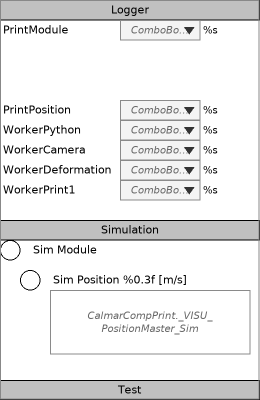
VISUALIZATION _VISU_Pm_Maxliner_Debug  // 260x400
VAR_IN_OUT
	mInst : FB_PrintModule_Maxliner;
END_VAR
    Rectangle (0,220 260x20), "Simulation"
    Ellipse (20,270 20x20), tooltip "Sim position"
        toggle mInst.fbPrintPosition._bSim
    Rectangle (50,270 200x20), "Sim Position %0.3f [m/s]", text variable: mInst.fbPrintPosition.fbPositionMaster._fSimSpeed
        OnMouseClick: write the text variable via Default
    Rectangle (0,0 260x20), "Logger"
    Rectangle (0,100 120x20), "PrintPosition"
    Rectangle (200,100 60x20), "%s", tooltip "LogLevel", text variable: mInst.fbPrintPosition._loglevel
        OnMouseClick: write the text variable via Default
    Rectangle (0,140 120x20), "WorkerCamera"
    Rectangle (200,140 60x20), "%s", tooltip "LogLevel", text variable: mInst.fbWorkerCamera._loglevel
        OnMouseClick: write the text variable via Default
    Rectangle (0,180 120x20), "WorkerPrint1"
    Rectangle (200,180 60x20), "%s", tooltip "LogLevel", text variable: mInst.fbWorkerPrint[1]._loglevel
        OnMouseClick: write the text variable via Default
    Rectangle (0,160 120x20), "WorkerDeformation"
    Rectangle (200,160 60x20), "%s", tooltip "LogLevel", text variable: mInst.fbWorkerDeformation._loglevel
        OnMouseClick: write the text variable via Default
    ComboBoxInteger (120,180 80x20), tooltip "LogLevel", variable: mInst.fbWorkerPrint[1]._loglevel, text list: 'LogSeverity'
    ComboBoxInteger (120,160 80x20), tooltip "LogLevel", variable: mInst.fbWorkerDeformation._loglevel, text list: 'LogSeverity'
    ComboBoxInteger (120,140 80x20), tooltip "LogLevel", variable: mInst.fbWorkerCamera._loglevel, text list: 'LogSeverity'
    ComboBoxInteger (120,100 80x20), tooltip "LogLevel", variable: mInst.fbPrintPosition._loglevel, text list: 'LogSeverity'
    Frame (50,290 200x64)
        shows CalmarCompPrint._VISU_PositionMaster_Sim(mInst := mInst.fbPrintPosition.fbPositionMaster)
    Rectangle (0,380 260x20), "Test"
    Ellipse (0,240 20x20), tooltip "Sim position"
        toggle mInst.bSimEnable
    Rectangle (30,240 200x20), "Sim Module"
    Rectangle (0,20 120x20), "PrintModule"
    Rectangle (200,20 60x20), "%s", tooltip "LogLevel", text variable: mInst._loglevel
        OnMouseClick: write the text variable via Default
    ComboBoxInteger (120,20 80x20), tooltip "LogLevel", variable: mInst._loglevel, text list: 'LogSeverity'
    Rectangle (0,120 120x20), "WorkerPython"
    Rectangle (200,120 60x20), "%s", tooltip "LogLevel", text variable: mInst.fbWorkerPython._loglevel
        OnMouseClick: write the text variable via Default
    ComboBoxInteger (120,120 80x20), tooltip "LogLevel", variable: mInst.fbWorkerPython._loglevel, text list: 'LogSeverity'
END_VISUALIZATION

(* stored: Version 1.1.0.1, ProductVersion 3.1.4024.11
   Visu _VISU_Pm_Maxliner_Debug: Id {5e3506d2-ad91-469d-8da5-134e295b40ea} *)
